FUNCTION_BLOCK ConveyorLSC EXTENDS ConveyorSC
VAR_OUTPUT
	lifterError AT %I* : BOOL;
	
	extended AT %I* : BOOL;
	retracted AT %I* : BOOL;
END_VAR
VAR	
	lifterEnable AT %Q* : BOOL := TRUE;
	lifterDirection AT %Q* : BOOL; //FALSE = up, TRUE = down
	lifterPulse AT %Q* : BOOL;
	lifterReset AT %Q* : BOOL;
END_VAR
VAR	
	lifterMode : (HOLD, LIFTER_EXTEND, LIFTER_RETRACT); 
	lifterPulser : TP; //pulses are assumed to be low-high-low
END_VAR

SUPER^();

lifterOverride();

lifterSequence();

METHOD backward : BOOL
VAR_INPUT
END_VAR
END_METHOD

METHOD extend : BOOL
VAR_INPUT
END_VAR
lifterMode := LIFTER_EXTEND;
END_METHOD

METHOD forward : BOOL
VAR_INPUT
END_VAR
END_METHOD

METHOD PROTECTED lifterOverride : BOOL
VAR_INPUT
END_VAR
IF
	(extended AND lifterMode = LIFTER_EXTEND) OR
	(retracted AND lifterMode = LIFTER_RETRACT)
THEN
	lifterMode := HOLD;
END_IF
END_METHOD

METHOD PROTECTED lifterSequence : BOOL
VAR_INPUT
END_VAR
VAR
	nextOp, prevOp : INT;
END_VAR
lifterPulser(IN:= , PT:= pulseWidth, Q=> , ET=> );
lifterPulser.IN := 
	lifterEnable AND 
	NOT lifterError AND 
	NOT lifterReset AND 
	( (lifterMode = LIFTER_EXTEND AND NOT extended) OR (lifterMode = LIFTER_RETRACT AND NOT retracted) ) AND
	lifterPulser.Q; //self-ending pulse

lifterPulse := lifterPulser.Q AND lifterPulser.ET < pulseWidth/2;
END_METHOD

METHOD reset : BOOL
VAR_INPUT
END_VAR
position := 0;
velocity := velocity; //no change

extend();
END_METHOD

METHOD retract : BOOL
VAR_INPUT
END_VAR
lifterMode := LIFTER_RETRACT;
END_METHOD

END_FUNCTION_BLOCK

(* stored: Version 1.1.0.1, ProductVersion 3.1.4024.11
   POU ConveyorLSC: Id {173b778f-3776-40af-8508-b38536d46f28}, SpecialFunc None
   Folder Private: Id {1b9abd46-42b0-4c2d-9ec7-18746ee0f7b2}
   Folder Properties: Id {93e21bd6-da8f-4da1-a613-a243d3058f6d}
   Folder Unused: Id {6b06cd7b-bad2-42a7-a341-c31d884c0e98}
   Method backward: Id {9b6b33ef-d8d0-4585-a8ef-7138765c392c}
   Method extend: Id {7046fa8f-b472-4aea-b5d8-8074c56085a5}
   Method forward: Id {c6a7a924-0827-4d06-b3b0-f36f374d2fdf}
   Method lifterOverride: Id {198bdd4d-ea1c-45e4-87ce-e9d0ddee8d0e}
   Method lifterSequence: Id {1d38bec5-edaf-46fc-b976-a81837f7eb79}
   Method reset: Id {25d42f91-6e59-48bd-8845-da39fdd8a3bf}
   Method retract: Id {e039dd37-a39c-4d00-bbab-5a1c1b80e2eb} *)
